Universal Robots PolyScope program: matlabcontrol.urp

Program matlabcontrol (createdIn=1.8.11657.0 lastSavedIn=3.3.4.310 directory=/programs/robotvision installation=default robotSerialNumber=2017353993)
Calibrated DH parameters: a=[0.000164, -0.372614, -0.390071, 0.000067, 0.000035, 0]; d=[0.088949, -236.832261, 239.457522, -2.515251, 0.094878, 0.082509]; alpha=[1.570462, -0.000861, -0.0155, 1.570767, -1.57079, 0]; deltaTheta=[0.000015, 0.500831, -0.604847, 0.10386, 0.000033, 0.000067]
BeforeStart
  receive_data := [6,0,0,0,0,0,0]
  pi := 3.1415
  Move_To_Pos := p[0.5,0,0.2,pi,0,0]
  Script: movej([0.23,-1.57,-1.6,-1.52,1.57,-1.34],v=0.2)
  Script: movej(get_inverse_kin(Move_To_Pos),v=0.4)
  Call SubProgram_3
  Script: socket_open("172.20.13.1",30000)
  task := [0,0]
  coop := 0
  moving := 0
Robot Program (runOnlyOnce=false motionType=MoveJ speed=1.047198 acceleration=1.396263 recalculateMotions=false)
  SuppressedNode
    MoveJ speed 60 deg/s, acceleration 80 deg/s^2 (recalculateMotions=false)
      Waypoint Waypoint_1 (Relative): relativeFromPosition TCP in base x=416.871 y=-406.97 z=211.075 mm, rx=1.6627 ry=-1.7508 rz=0.7521 rad; joints [-27.823, -125.587, -73.499, -225.375, -46.749, 144.79] deg; TCP in base x=416.871 y=-406.97 z=211.075 mm, rx=1.6627 ry=-1.7508 rz=0.7521 rad; joints [-27.823, -125.587, -73.499, -225.375, -46.749, 144.79] deg; flange x=416.623 y=-407.059 z=211.624 mm, rx=1.6638 ry=-1.7496 rz=0.7522 rad
  SuppressedNode
    coop := 1
  SuppressedNode
    Wait Sleep waitTime=2
  SuppressedNode
    coop := 0
  Script: task=socket_read_ascii_float(1)
  If task[1]≟2
    Call SubProgram_2
    task := [0,0]
  ElseIf task[1]≟3
    coop := 1
    Script: teach_mode()
    Script: socket_send_string("1")
    task := [0,0]
  ElseIf task[1]≟4
    coop := 0
    Script: end_teach_mode()
    Script: socket_send_string("1")
    task := [0,0]
  ElseIf task[1]≟5
    Script: set_tool_digital_out(0, True )
    Script: socket_send_string("1")
    task := [0,0]
  ElseIf task[1]≟6
    Script: set_tool_digital_out(0, False )
    Script: socket_send_string("1")
    task := [0,0]
  ElseIf task[1]≟1
    Call SubProgram_1
  Wait Sleep waitTime=0.01
Thread Thread_1 (runOnlyOnce=false trackProgramExecution=false)
  If coop≟1
    Loop While (checkContinuously=false) expression=coop≟1
      SuppressedNode
        Force Frame feature=Base; selection=[1, 1, 1, 1, 1, 1]; wrench=[0, 0, 0, 0, 0, 0]; limitsForce=[0.15, 0.15, 0.15, 1.047198, 1.047198, 1.047198]; limitsMotion=[0.1, 0.1, 0.1, 0.174533, 0.174533, 0.174533]
          Wait Sleep waitTime=0.01
      Wait Sleep waitTime=0.01
    coop := 0
    Call SubProgram_3
  Else 
    Script: movel(Move_To_Pos,a=0.4,v=0.4,r=0)
    If moving≟1
      Wait Sleep waitTime=0.05
      Script: socket_send_string("X")
      moving := 0
    Wait Sleep waitTime=0.01
SubProgram -> SubProgram_1
SubProgram -> SubProgram_2
SubProgram -> SubProgram_3
SubProgram SubProgram_3 (keepSynchronizedWithDisk=false trackProgramExecution=false)
  Script: pose_1=get_forward_kin()
  pointer := 0
  Loop While (checkContinuously=false) expression=pointer<receive_data[0]
    Script: Move_To_Pos[pointer]=pose_1[pointer]
    pointer := pointer+1
SubProgram SubProgram_2 (keepSynchronizedWithDisk=false trackProgramExecution=false)
  Script: pose_1=get_forward_kin()
  Script: socket_send_string(pose_1)
SubProgram SubProgram_1 (keepSynchronizedWithDisk=false trackProgramExecution=false)
  Script: receive_data=socket_read_ascii_float(6)
  If receive_data[0]≠6
    Script: socket_send_string("0")
  Else 
    Script: socket_send_string("1")
    pointer := 0
    Loop While (checkContinuously=false) expression=pointer<receive_data[0]
      Script: Move_To_Pos[pointer]=receive_data[pointer+1]
      pointer := pointer+1
    task := [0,0]
    moving := 1
